FUNCTION_BLOCK Stage1 (* Template for a Basic Function Block Type *)
  (* Standard: 61499-2 *)
  (* Version 1.0, 2021-06-20, HP *)
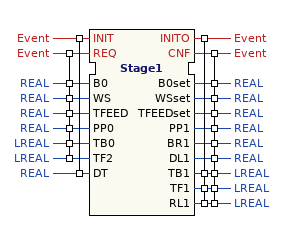
  EVENT_INPUT
    INIT WITH DT; (* Initialization Request *)
    REQ WITH B0, WS, TFEED, PP0, TB0, TF2; (* Normal Execution Request *)
  END_EVENT
  EVENT_OUTPUT
    INITO WITH TB1, TF1, RL1; (* Initialization Confirm *)
    CNF WITH PP1, BR1, TB1, DL1, TF1, B0set, WSset, TFEEDset, RL1; (* Execution Confirmation *)
  END_EVENT
  VAR_INPUT
    B0 : REAL; (* Input event qualifier *)
    WS : REAL;
    TFEED : REAL;
    PP0 : REAL;
    TB0 : LREAL;
    TF2 : LREAL;
    DT : REAL;
  END_VAR
  VAR_OUTPUT
    B0set : REAL;
    WSset : REAL;
    TFEEDset : REAL;
    PP1 : REAL;
    BR1 : REAL;
    DL1 : REAL;
    TB1 : LREAL;
    TF1 : LREAL;
    RL1 : LREAL;
  END_VAR
  VAR
    AB : REAL; (* Internal Variabel *)
    UU : REAL; (* Internal Variabel *)
    TREF : REAL; (* Internal Variabel *)
    AD : REAL; (* Internal Variabel *)
    AHC : REAL; (* Internal Variabel *)
    AHR : REAL; (* Internal Variabel *)
    AS : REAL; (* Internal Variabel *)
    REC : REAL; (* Internal Variabel *)
    WN : REAL; (* Internal Variabel *)
    WN_1 : REAL; (* Internal Variabel *)
    XKN : REAL; (* Internal Variabel *)
    C1 : REAL; (* Internal Variabel *)
    HS : REAL; (* Internal Variabel *)
    G : REAL; (* Internal Variabel *)
    W1 : REAL; (* Internal Variabel *)
    TFREC : REAL; (* Internal Variabel *)
    TS : REAL; (* Internal Variabel *)
    DTS : REAL; (* Internal Variabel *)
    TF1_last : REAL; (* Internal Variabel *)
    TF2_last : REAL; (* Internal Variabel *)
    RL1_last : REAL; (* Internal Variabel *)
    TB1_last : REAL; (* Internal Variabel *)
    USS : REAL; (* Internal Variabel *)
    RHOB : REAL; (* Internal Variabel *)
    CPB : REAL; (* Internal Variabel *)
    CPF : REAL; (* Internal Variabel *)
    FMW : REAL; (* Internal Variabel *)
    HLV : REAL; (* Internal Variabel *)
    HV : REAL; (* Internal Variabel *)
    BPR : REAL; (* Internal Variabel *)
    FMC : REAL; (* Internal Variabel *)
    U : REAL; (* Internal Variabel *)
    A : REAL; (* Internal Variabel *)
    B : REAL; (* Internal Variabel *)
    C : REAL; (* Internal Variabel *)
    a : REAL;
    p : REAL;
    q : REAL;
    b : REAL;
    l : REAL;
    D1 : REAL; (* Internal Variabel *)
    TC : REAL; (* Internal Variabel *)
    PC : REAL; (* Internal Variabel *)
    DTB0 : REAL; (* Internal Variabel *)
    DEN0 : REAL; (* Internal Variabel *)
    DTB1 : REAL; (* Internal Variabel *)
    DEN1 : REAL; (* Internal Variabel *)
    d : REAL;
    A1 : REAL;
    A2 : REAL;
    A3 : REAL;
    A4 : REAL;
    A5 : REAL;
    A6 : REAL;
    DH1 : REAL; (* Internal Variabel *)
    DP1 : REAL; (* Internal Variabel *)
    DPDH1 : REAL; (* Internal Variabel *)
    m : REAL;
    n : REAL;
    DT1 : REAL; (* Internal Variabel *)
    VR1 : REAL; (* Internal Variabel *)
    DELTA1 : REAL;
    DELTA45 : REAL; (* Internal Variabel *)
    DELTA23 : REAL; (* Internal Variabel *)
    DELTA1_last : REAL; (* Internal Variabel *)
    DELTA23_last : REAL; (* Internal Variabel *)
    DELTA45_last : REAL; (* Internal Variabel *)
  END_VAR
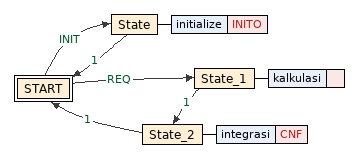
  EC_STATES
    START; (* Initial State *)
    State : initialize -> INITO;
    State_1 : kalkulasi;
    State_2 : integrasi -> CNF;
  END_STATES
  EC_TRANSITIONS
    START TO State := INIT;
    State TO START := 1;
    START TO State_1 := REQ;
    State_1 TO State_2 := 1;
    State_2 TO START := 1;
  END_TRANSITIONS
  ALGORITHM initialize IN ST: (* Initialization algorithm *)
TREF :=273.15;
AB :=57.2727;
AHC :=4069.2;
AHR :=2639.7;
AS :=3225.7;
REC :=0.0;
//TF2:=TF2;

//TFEED :=TFEED1+TREF;
 //TS:=TS1+TREF;
WN :=3.0;
XKN :=0.68;
HS:=0.11;
G :=9.81;
W1 :=0.50;

   //initial condition
RL1:=0.520814850809769;
TB1 :=363.700385920319;
TF1 :=359.946661638812;
TF2:=357.473636725142;


TFREC :=  314.548634310388;

RL1_last :=RL1;
TB1_last :=TB1;
TF1_last :=TF1;
  END_ALGORITHM
  ALGORITHM kalkulasi IN ST: (* perhitungan *)
UU :=TFEED ;
U :=UU;

USS :=49.767;
C1 :=0.625;
RHOB :=1032.4; //maassa jenis brine
CPB :=1.00; //heatcapacity Brine
CPF :=1.00; //heat capacity feed
FMW :=23654.0;
HLV :=563.7959;
HV :=625.1971;
BPR :=2.192;
FMC :=34736.09;
//U :=UU; //feed temp



///  Calculate the physical properties

//A :=3.2437814;
//B :=5.86826*0.001;
//C :=1.1702379*0.00000001;
//D1 :=2.1878462*0.001;
//TC :=647.27;
//PC :=218.167;

//DTB0 :=TC-TB0;
//DEN0 :=(A+B*DTB0+C*DTB0*DTB0*DTB0)/(1+D1*DTB0)*DTB0/TB0;
//b:=DEN0;
//a:=10.0;
//PP0 :=PC/(EXPT(a, b));

A1 :=3.2437814;
A2:=5.86826*0.001;
A3:=1.1702379*0.00000001;
A4 :=2.1878462*0.001;
A5 :=647.27;
A6 :=218.167;

DTB1 :=A5-TB1;
DEN1 :=(A1+A2*DTB1+A3*DTB1*DTB1*DTB1)/(1+A4*DTB1)*DTB1/TB1;
p:=DEN1;
q:=10.0;
PP1 :=A6/(EXPT(q, p));

// calculate the brine flow rates
DP1:=PP0-PP1;
DH1:=RL1-C1*HS;
DPDH1 :=DP1*101000+G*RHOB*DH1;
m:=DPDH1*RHOB;
n:=0.5;
BR1 :=WN*XKN*RL1*(EXPT(m, n));
BR1 :=BR1*60.0/1000.0;

// calculate the vapor flow rates

DT1 :=TB1-BPR/1.8-(TF2+TF1)*0.5;
VR1 :=U*AHC*DT1/HLV/1000.0;
DL1 :=VR1;


//// state equation
DELTA1 :=(B0-BR1-VR1)*1000.0/RHOB/AB;
DELTA23 :=(B0*CPB*(TB0-TB1));
DELTA23 :=DELTA23-VR1*(HV-CPB*(TB1-TREF));
DELTA23 :=DELTA23*1000.0/AB/RHOB/CPB/RL1;

DELTA45 :=B0*CPF*(TF2-TF1)*1000;
DELTA45 :=DELTA45+(U*AHC*DT1);
DELTA45 :=DELTA45/FMW/CPF;
  END_ALGORITHM
  ALGORITHM integrasi IN ST: (* algoritma integrasi *)
B0set:=B0;
WSset:=WS ;
TFEEDset:=TFEED;
//integrasi
RL1 := (DELTA1 + DELTA1_last)*0.5*DT + RL1_last;
DELTA1_last :=DELTA1 ;
RL1_last :=RL1;

TB1 :=(DELTA23 + DELTA23_last)*0.5*DT + TB1_last;
DELTA23_last :=DELTA23 ;
TB1_last:=TB1;

TF1 := (DELTA45 + DELTA45_last)*0.5*DT + TF1_last;
DELTA45_last :=DELTA45 ;
TF1_last :=TF1;
  END_ALGORITHM
END_FUNCTION_BLOCK
